TYPE ST_AxisFault :
STRUCT
	bMcPowerOff		: BOOL;
	bOverCurrent	: BOOL;
	bSTO			: BOOL;
END_STRUCT
END_TYPE

(* stored: Version 1.1.0.1, ProductVersion 3.1.4024.12
   DUT ST_AxisFault: Id {bd4f618b-a43e-4fc3-90c9-37ced9f55beb} *)
